PROGRAM main
VAR
	CoolingPumpStatus AT %QX0.0 : bool;
	CurrentTemp AT %MW0 : int := 0;
	MaxLimitTemp AT %MW1 : int := 50;
END_VAR

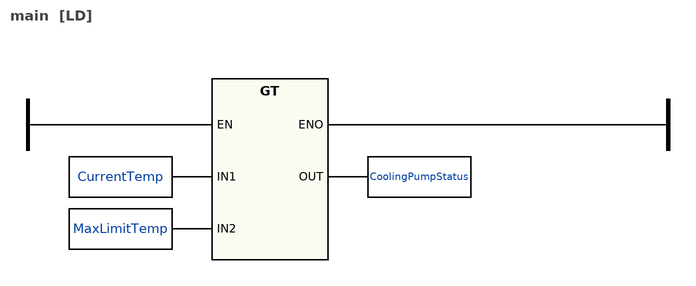
(* LD diagram, written out as Structured Text *)
CoolingPumpStatus := CurrentTemp > MaxLimitTemp;
END_PROGRAM
